FUNCTION_BLOCK FB_FastCounter
VAR_IN_OUT
	PulseCount : UDINT;
END_VAR
VAR_INPUT
	FlowSensor : BOOL;
END_VAR
VAR
	testclk : TON; // testclk
	
	rtPulse : R_TRIG; // Edge detection
END_VAR

// Look for the "False -> True" transition
rtPulse(CLK := FlowSensor);

//testclk(IN := NOT testclk.Q, PT := T#50ms);
// If edge detected, increment the global counter
IF rtPulse.Q THEN
    PulseCount := PulseCount + 1;
END_IF
	
//IF testclk.Q THEN
//	PulseCount := PulseCount + 1;
//END_IF

END_FUNCTION_BLOCK

(* stored: Version 1.1.0.1
   POU FB_FastCounter: Id {e3335d9d-e004-497a-b538-416b95187f0d}, SpecialFunc None *)
